{attribute 'qualified_only'}
{attribute 'strict'}
{attribute 'to_string'}
TYPE E_EmergencyReason : 
(
	ERR_NONE 			:= 0,
	ERR_HearBeatFail 	:= 1,
	ERR_EmergencyOverGS := 2,
	ERR_IMD 			:= 3,
	ERR_BMS 			:= 4,
	ERR_CHECKCRITICAL	:= 5
);
END_TYPE

(* stored: Version 1.1.0.1
   DUT E_EmergencyReason: Id {3a4d48bd-7fd6-4037-8525-5168b2f447bf} *)
